FUNCTION_BLOCK Automatic
VAR_INPUT
END_VAR
VAR_OUTPUT
END_VAR
VAR
	inputPiston: PistonInputLogic;
	outputPiston: PistonOutputLogic;
	tablelogic: TableLogic;
END_VAR

inputPiston();
tableLogic();
outputPiston();

IF gvl.FotocellOutput THEN
	gvl.MotorBeltMove := FALSE;
END_IF

END_FUNCTION_BLOCK

(* stored: Version 1.1.0.1, ProductVersion 3.1.4024.12
   POU Automatic: Id {f92e9b7a-f792-439f-a45d-f4a06f7fc726}, SpecialFunc None *)
